FUNCTION_BLOCK FB_PROCESS_MAIN IMPLEMENTS I_PROCESS_MAIN
VAR //General
	{attribute 'instance-path'} 
  {attribute 'noinit'} 
	strInstancePath:									                      STRING;
	bInit: 												                          BOOL:=TRUE;
	strFullObjectPath: 								                      STRING;
	stEvent:											                          ST_EVENT;
	bAck:												                            BOOL;
	bNext:                                                  BOOL;
  bStop:                                                  BOOL;
END_VAR
VAR   // From FB_init	
	itfLogEvents: 										                      I_HANDLE_EVENTS;
  itfOpMode:											                        I_OP_MODE;  
  itfTimerNest1:                                          I_CLOCK; 
  itfTimerNest2:                                          I_CLOCK; 
  itfTimerNest3:                                          I_CLOCK; 
  itfTimerNest4:                                          I_CLOCK;
  itfNest1:                                               I_PROCESS_NEST1;
  itfNest2:                                               I_PROCESS_NEST2_4;
  itfNest3:                                               I_PROCESS_NEST2_4;
  itfNest4:                                               I_PROCESS_NEST2_4;
  itfLowPressurePump:                                     I_PUMP_WITH_BYPASS;
  itfOilCooler:                                           I_PUMP;
  itfBypassPump:                                          I_PUMP;
  itfLevelSwitch_AggregateTank1_Out1:                     I_BINARY_SWITCH;
  itfLevelSwitch_AggregateTank1_Out2:                     I_BINARY_SWITCH;
  itfTemperatureSwitch_AggregateTank1_Out1:               I_BINARY_SWITCH;
  itfTemperatureSwitch_AggregateTank1_Out2:               I_BINARY_SWITCH;
  itfLevelSwitch_AggregateTank2_Out1:                     I_BINARY_SWITCH;
  itfLevelSwitch_AggregateTank2_Out2:                     I_BINARY_SWITCH;
  itfLevelSwitch_AggregateTank2_Out3:                     I_BINARY_SWITCH;
  itfSwitch_AggregateFilter_Dirty:                        I_BINARY_SWITCH;  
END_VAR                                      				
VAR	// Step chain control                				
  eSeq, eLastSeq, eNextSeq:					                      E_SEQ_PROCESS; 
                  				
  //eActiveSeqState, eLastActiveSeqState:                 E_SEQ_GENERAL;
	(*
  iInternalSeqStateCase, iLastInternalSeqStateCase:       INT:=0;       
	tonDelay, tonTimeOut, tonStepTime:						          TON;
	tDelay:													                        TIME := T#100MS;
	tTimeOut:												                        TIME := T#100MS;
	tTimeOutExt:											                      TIME := T#100MS;
	bDelayActive, bTimeOutActiveQuit, bTimeOutActiveNoQuit:	BOOL;//Timer Option
	bActiveStep, bDebugAcitve, bDebugNext:					        BOOL;//Debug Option
	i:														                          INT;
 	iError:													                        INT; //ERROR-CODE                    	                   		
	listLastSteps:											                    ARRAY[0..49] OF ST_LAST_STEPS;	
	strExtraInfo:											                      STRING; 
	eStep_Type:												                      E_STEP_STATE_TYPE; 
	bDebugModeActive:										                    BOOL;   
	bWaitForBreakpoint:										                  BOOL;
	bBreakpointActive:										                  BOOL;
	bDebugResume:											                      BOOL;   
	listBreakpoint:											                    ARRAY[0..10] OF  INT;    
  *)
  i:														                            INT;
  stSeqCtrlGeneral:											                    ST_SEQ_CTRL_GEN;  
  strSeq:                                                   STRING;   	
  uiRequestId:                                              UINT;
END_VAR                                             		
VAR                                                 		
	bMethodeFromExtStarted:									                BOOL;
	bMethodeFromExtActive:									                BOOL;
	bMethodeFromExtDone:									                  BOOL;
	strTemp:												                        STRING;
END_VAR   
VAR
  udiCurrentCyclesNest1:                                  UDINT := 0;
  udiCurrentCyclesNest2:                                  UDINT := 0;
  udiCurrentCyclesNest3:                                  UDINT := 0;
  udiCurrentCyclesNest4:                                  UDINT := 0;
  udiCyclesPerLoop:                                       UDINT := 0;
  udiLoops:                                               UDINT := 0;
  uiCurrentLoop:                                          UINT := 1;
  udiResidualVal:                                         UDINT := 0;
  uiVentCount:                                            UINT;
  iOpStep:                                                INT := 0;
  bRunning:                                               BOOL;
END_VAR 
VAR // Input variables
  stERParams:                                             ST_RECIPE_ENDURANCE_RUN;
  stBPDParams:                                            ST_RECIPE_BREAK_PRESSURE;
  stLT1Params:                                            ST_RECIPE_LEAK_TEST1;
  stLT2Params:                                            ST_RECIPE_LEAK_TEST2;
END_VAR                   	
VAR_TEMP                    	
	iTemp:											                            INT;
END_VAR

// Set FBs and Interfaces ready after switch internal step
IF stSeqCtrlGeneral.iInternalSeqStateCase <> stSeqCtrlGeneral.iLastInternalSeqStateCase AND NOT stSeqCtrlGeneral.bExitSetReadyState THEN
  IF TRUE
  AND itfNest1.M_SetReady()
  AND itfNest2.M_SetReady()
  AND itfNest3.M_SetReady()
  AND itfNest4.M_SetReady()
  AND itfLowPressurePump.M_SetReady()
  AND itfOilCooler.M_SetReady()
  AND itfBypassPump.M_SetReady()
  THEN
    stSeqCtrlGeneral.bExitSetReadyState := TRUE;
  ELSE
    RETURN;
  END_IF
END_IF

stSeqCtrlGeneral.strObject:=F_CreateObjectName(strInstancePath);

// First method call
_m_SequenceManager();
//_m_SaveLastStep();

strSeq := TO_STRING(eSeq);

CASE eSeq OF 
  E_SEQ_VALVE.BASE:;
  
	E_SEQ_PROCESS.INIT: _m_Seq_INIT();
		IF TRUE
		AND (stSeqCtrlGeneral.eActiveSeqState = E_SEQ_GENERAL.DONE) 
		THEN
      eSeq := eNextSeq := E_SEQ_PROCESS.BASE;
		END_IF
		
	E_SEQ_PROCESS.SETUP:;
  
	// Process
	E_SEQ_PROCESS.ENDURANCE_RUN: _m_Seq_ENDURANCE_RUN();
    IF TRUE
		AND (stSeqCtrlGeneral.eActiveSeqState = E_SEQ_GENERAL.DONE) 
		THEN
      eSeq := eNextSeq := E_SEQ_PROCESS.BASE;
		END_IF
 
  E_SEQ_PROCESS.BREAK_PRESSURE_DET: _m_Seq_BREAK_PRESSURE_DET();
    IF TRUE
		AND (stSeqCtrlGeneral.eActiveSeqState = E_SEQ_GENERAL.DONE) 
		THEN
      eSeq := eNextSeq := E_SEQ_PROCESS.BASE;
		END_IF
    
  E_SEQ_PROCESS.LEAK_TEST_1: _m_Seq_LEAK_TEST_1();
    IF TRUE
		AND (stSeqCtrlGeneral.eActiveSeqState = E_SEQ_GENERAL.DONE) 
		THEN
      eSeq := eNextSeq := E_SEQ_PROCESS.BASE;
		END_IF
    
  E_SEQ_PROCESS.LEAK_TEST_2: _m_Seq_LEAK_TEST_2();
    IF TRUE
		AND (stSeqCtrlGeneral.eActiveSeqState = E_SEQ_GENERAL.DONE) 
		THEN
      eSeq := eNextSeq := E_SEQ_PROCESS.BASE;
		END_IF
       
  E_SEQ_PROCESS.STOP: _m_Seq_STOP();
    IF TRUE
		AND (stSeqCtrlGeneral.eActiveSeqState = E_SEQ_GENERAL.DONE) 
		THEN
      eSeq := eNextSeq := E_SEQ_PROCESS.BASE;
		END_IF
    
  E_SEQ_PROCESS.STOP_ENGINE: _m_Seq_STOP_ENGINE();
    IF TRUE
		AND (stSeqCtrlGeneral.eActiveSeqState = E_SEQ_GENERAL.DONE) 
		THEN
      eSeq := eNextSeq := E_SEQ_PROCESS.BASE;
		END_IF
    
  E_SEQ_PROCESS.ESTOP: _m_Seq_ESTOP();
    IF TRUE
		AND (stSeqCtrlGeneral.eActiveSeqState = E_SEQ_GENERAL.DONE) 
		THEN
      eSeq := eNextSeq := E_SEQ_PROCESS.BASE;
		END_IF
  
  // End
	E_SEQ_PROCESS.END:;
	E_SEQ_PROCESS.ERROR_SEQ:;	
END_CASE

strTemp:=TO_STRING(eSeq);

METHOD PRIVATE _m_DebugManager
VAR_INPUT
	iStepID: int;
END_VAR
IF TRUE
AND THIS^.stSeqCtrlGeneral.bDebugModeActive 
AND NOT THIS^.stSeqCtrlGeneral.bActiveStep
THEN


THIS^.stSeqCtrlGeneral.bBreakpointActive:=FALSE;

FOR i:=0 TO 10 DO
	
	IF TRUE
	AND iStepID=THIS^.stSeqCtrlGeneral.listBreakpoint[i] 
	AND iStepID<>0
	THEN
		EXIT;
	END_IF
END_FOR
IF (i<=10) THEN
	THIS^.stSeqCtrlGeneral.bBreakpointActive:=TRUE;
END_IF

END_IF
END_METHOD

METHOD _m_Delay : BOOL
VAR_INPUT
	DelayTime:	TIME;
END_VAR
THIS^.stSeqCtrlGeneral.bDelayActive:=TRUE;
THIS^.stSeqCtrlGeneral.tDelay:=DelayTime;
_m_Delay:=FALSE;
IF THIS^.stSeqCtrlGeneral.tonDelay.Q THEN
	_m_Delay:=TRUE;
END_IF
END_METHOD

METHOD PRIVATE _m_GeneralStepSetting : BOOL
VAR_INPUT
	StepType:			    	E_STEP_STATE_TYPE;
	InfoTextID:					STRING(20);
	EnableDebug:	   			BOOL;	
	
END_VAR
IF THIS^.stSeqCtrlGeneral.bActiveStep THEN
	THIS^.stSeqCtrlGeneral.eStep_Type:=StepType;
	THIS^.stSeqCtrlGeneral.strExtraInfo:= GenLib.F_RET_TXTLIST_ENTRY(strPortNr:='851',strID:='',strTxtLstName:=InfoTextID);
END_IF
END_METHOD

METHOD PRIVATE _m_SaveLastStep : BOOL
VAR_INPUT
END_VAR
VAR
	i: dint;
END_VAR
IF NOT THIS^.stSeqCtrlGeneral.bActiveStep THEN
	
	FOR i:=49 TO 1 BY -1 DO
			stSeqCtrlGeneral.listLastSteps[i].strStepName:=stSeqCtrlGeneral.listLastSteps[i-1].strStepName;
			stSeqCtrlGeneral.listLastSteps[i].tStepTime:=stSeqCtrlGeneral.listLastSteps[i-1].tStepTime;
			stSeqCtrlGeneral.listLastSteps[i].tDelayTime:=stSeqCtrlGeneral.listLastSteps[i-1].tDelayTime;
	END_FOR
	stSeqCtrlGeneral.listLastSteps[0].strStepName:=TO_STRING(THIS^.eSeq);
	stSeqCtrlGeneral.listLastSteps[1].tStepTime:=THIS^.stSeqCtrlGeneral.tonStepTime.ET;
	stSeqCtrlGeneral.listLastSteps[1].tStepTime:=THIS^.stSeqCtrlGeneral.tonDelay.ET;
ELSE
	stSeqCtrlGeneral.listLastSteps[0].tStepTime:=THIS^.stSeqCtrlGeneral.tonStepTime.ET;
	stSeqCtrlGeneral.listLastSteps[0].tDelayTime:=THIS^.stSeqCtrlGeneral.tonDelay.ET;	
END_IF
END_METHOD

METHOD PRIVATE _m_Seq_BREAK_PRESSURE_DET : E_SEQ_PROCESS
VAR_INPUT
END_VAR
VAR
	ActiveSeq: STRING;
END_VAR
VAR
	
END_VAR
//THIS^._m_GeneralStepSetting(StepType:=E_STEP_STATE_TYPE.INIT,
ActiveSeq := TO_STRING(THIS^.eSeq);

CASE THIS^.stSeqCtrlGeneral.eActiveSeqState OF
E_SEQ_GENERAL.READY:;

	
E_SEQ_GENERAL.EXECUTE:;
	IF TRUE
	THEN
		THIS^.stSeqCtrlGeneral.eActiveSeqState := E_SEQ_GENERAL.RESET;
	END_IF
E_SEQ_GENERAL.RESET:;
	stSeqCtrlGeneral.iInternalSeqStateCase := 0;
	IF TRUE
	THEN
		THIS^.stSeqCtrlGeneral.eActiveSeqState := E_SEQ_GENERAL.BUSY;
	END_IF
  
E_SEQ_GENERAL.BUSY:;
	CASE THIS^.stSeqCtrlGeneral.iInternalSeqStateCase OF
    0:  // check validity
      IF TRUE
      AND THIS^.stBPDParams.rMinSpeedInMmPerS > 0.1
      AND THIS^.stBPDParams.rEndPosTol > 0
      AND THIS^.stBPDParams.rIncreaseInterval > 0.1
      AND THIS^.stBPDParams.rIncreaseInterval < 10
      AND THIS^.stBPDParams.rNokLimit > 1
			THEN 
				THIS^.stSeqCtrlGeneral.iInternalSeqStateCase := 5; 
      ELSE
        THIS^.stSeqCtrlGeneral.eActiveSeqState := E_SEQ_GENERAL.ERROR; // Error step
			END_IF
      
    5:  // Start timer
      IF THIS^.itfNest1.P_EnableState THEN
        THIS^.itfTimerNest1.M_StartTimer();
			END_IF
      THIS^.stSeqCtrlGeneral.iInternalSeqStateCase := 10;

    10:  // Nest 1 vent cylinder
      IF TRUE
      AND THIS^.itfLowPressurePump.M_Bypass(bEnable:= TRUE)
			AND THIS^.itfNest1.M_VentCylinder(uiVentCount:= THIS^.stBPDParams.uiVentCycles)
			THEN 
				THIS^.stSeqCtrlGeneral.iInternalSeqStateCase := 20; 
			END_IF
      
    20:  // Low pressure pump off
      IF TRUE  
      AND THIS^.itfLowPressurePump.M_Off()
			THEN 
				THIS^.stSeqCtrlGeneral.iInternalSeqStateCase := 30; 
			END_IF
      
    30:  // Nest 1 determinate stroke length
      IF TRUE 
			AND THIS^.itfNest1.M_MeasureStrokeLength()
			THEN 
				THIS^.stSeqCtrlGeneral.iInternalSeqStateCase := 40; 
			END_IF
      
    40:  // Nest 1 endurance run
      IF TRUE 
			AND THIS^.itfNest1.M_BreakPressureDet(stBreakPressureParams:= THIS^.stBPDParams)
			THEN 
				THIS^.stSeqCtrlGeneral.iInternalSeqStateCase := 1000; // Exit step
			END_IF
      
    1000: // Exit step
      IF TRUE 
      AND THIS^.itfTimerNest1.M_StopTimer()
			THEN 
				THIS^.stSeqCtrlGeneral.iInternalSeqStateCase := 9999; 
			END_IF
      
	ELSE
		THIS^.stSeqCtrlGeneral.eActiveSeqState := E_SEQ_GENERAL.DONE;  
	END_CASE
	THIS^.stSeqCtrlGeneral.strExtraInfo := CONCAT('Internal state: ', TO_STRING(THIS^.stSeqCtrlGeneral.iInternalSeqStateCase));
E_SEQ_GENERAL.DONE:;
E_SEQ_GENERAL.ERROR:;
E_SEQ_GENERAL.TIME_OUT:; 

IF TRUE
AND THIS^.stSeqCtrlGeneral.bTimeOutActiveQuit 
THEN
  THIS^.stSeqCtrlGeneral.strExtraInfo := 'Bitte quittieren und erneut testen';
  IF TRUE
  //AND itfOpMode.P_QUIT
  THEN
    THIS^.stSeqCtrlGeneral.eActiveSeqState := E_SEQ_GENERAL.EXECUTE;
	END_IF
  
END_IF

ELSE
  THIS^.stSeqCtrlGeneral.eActiveSeqState := E_SEQ_GENERAL.ERROR;
END_CASE
END_METHOD

METHOD PRIVATE _m_Seq_ENDURANCE_RUN : E_SEQ_PROCESS
VAR_INPUT
END_VAR
VAR
	ActiveSeq:                      STRING;
END_VAR
//THIS^._m_GeneralStepSetting(StepType:=E_STEP_STATE_TYPE.INIT,
ActiveSeq := TO_STRING(THIS^.eSeq);

CASE THIS^.stSeqCtrlGeneral.eActiveSeqState OF
E_SEQ_GENERAL.READY:;

	
E_SEQ_GENERAL.EXECUTE:;
	IF TRUE
	THEN
		THIS^.stSeqCtrlGeneral.eActiveSeqState := E_SEQ_GENERAL.RESET;
	END_IF
E_SEQ_GENERAL.RESET:;
	stSeqCtrlGeneral.iInternalSeqStateCase := 0;
	IF TRUE
	THEN
    THIS^.udiCyclesPerLoop := THIS^.stERParams.udiCycles;
    THIS^.udiLoops := 1;
    THIS^.uiCurrentLoop := 1;
    THIS^.udiResidualVal := 0;
		THIS^.stSeqCtrlGeneral.eActiveSeqState := E_SEQ_GENERAL.BUSY;
	END_IF
  
E_SEQ_GENERAL.BUSY:;
	CASE THIS^.stSeqCtrlGeneral.iInternalSeqStateCase OF
    0:  // check validity
      IF TRUE
      AND THIS^.stERParams.rSpeedA > 1
      AND THIS^.stERParams.rSpeedB > 1
      AND THIS^.stERParams.rTurningPointHP > 0
      AND THIS^.stERParams.rTurningPointWP > 0
      AND THIS^.stERParams.rWorkForceA > 0.1
      AND THIS^.stERParams.rWorkForceB > 0.1
      AND THIS^.stERParams.udiCycles > 1
			THEN 
				THIS^.stSeqCtrlGeneral.iInternalSeqStateCase := 5; 
      ELSE
        THIS^.stSeqCtrlGeneral.eActiveSeqState := E_SEQ_GENERAL.ERROR; // Error step
			END_IF
      
    5:  // Start timer
      IF THIS^.itfNest1.P_EnableState THEN
        THIS^.itfTimerNest1.M_StartTimer();
			END_IF
      IF THIS^.itfNest2.P_EnableState THEN
        THIS^.itfTimerNest2.M_StartTimer();
			END_IF
      IF THIS^.itfNest3.P_EnableState THEN
        THIS^.itfTimerNest3.M_StartTimer();
			END_IF
      IF THIS^.itfNest4.P_EnableState THEN
        THIS^.itfTimerNest4.M_StartTimer();
			END_IF
      THIS^.stSeqCtrlGeneral.iInternalSeqStateCase := 10;

    10:  // Nest 1-4 vent cylinder
      IF TRUE
      AND THIS^.itfLowPressurePump.M_Bypass(bEnable:= TRUE)
			AND THIS^.itfNest1.M_VentCylinder(uiVentCount:= THIS^.stERParams.uiVentCycles)
      AND THIS^.itfNest2.M_VentCylinder(uiVentCount:= THIS^.stERParams.uiVentCycles)
      AND THIS^.itfNest3.M_VentCylinder(uiVentCount:= THIS^.stERParams.uiVentCycles)
      AND THIS^.itfNest4.M_VentCylinder(uiVentCount:= THIS^.stERParams.uiVentCycles)
			THEN 
				THIS^.stSeqCtrlGeneral.iInternalSeqStateCase := 20; 
			END_IF
      
    20:  // Nest 1-4 determinate stroke length
      IF TRUE  
      AND THIS^.itfLowPressurePump.M_On()
			AND THIS^.itfNest1.M_MeasureStrokeLength()
      AND THIS^.itfNest2.M_MeasureStrokeLength()
      AND THIS^.itfNest3.M_MeasureStrokeLength()
      AND THIS^.itfNest4.M_MeasureStrokeLength()
			THEN 
				THIS^.stSeqCtrlGeneral.iInternalSeqStateCase := 30; 
			END_IF
      
    30:  // Nest 1 determinate max speed (VMAX)
      IF TRUE  
			AND THIS^.itfNest1.M_MaxSpeedRecord(stEnduranceRunParams:= THIS^.stERParams)
			THEN 
        IF TRUE
        AND (THIS^.stERParams.rSpeedA > THIS^.itfNest1.P_MaxSpeedInMmPerSWP * THIS^.itfNest1.P_SpeedEfficiencyFactor
        OR THIS^.stERParams.rSpeedB > THIS^.itfNest1.P_MaxSpeedInMmPerSHP * THIS^.itfNest1.P_SpeedEfficiencyFactor) 
        THEN
          THIS^.itfNest2.M_SetEnableState(bEnable:= FALSE);
          THIS^.itfNest3.M_SetEnableState(bEnable:= FALSE);
          THIS^.itfNest4.M_SetEnableState(bEnable:= FALSE);
          THIS^.itfTimerNest2.M_StopTimer();
          THIS^.itfTimerNest3.M_StopTimer();
          THIS^.itfTimerNest4.M_StopTimer();
				END_IF
				THIS^.stSeqCtrlGeneral.iInternalSeqStateCase := 40; 
			END_IF
      
    40:  // Calc loops and cycles
      IF TRUE
      AND THIS^.stERParams.bEnableLeakTest1
      THEN
        THIS^.udiCyclesPerLoop := THIS^.stERParams.udiLT1_Interval;
        THIS^.udiLoops := THIS^.stERParams.udiCycles / THIS^.stERParams.udiLT1_Interval - 1;
        THIS^.udiResidualVal := THIS^.stERParams.udiCycles - THIS^.udiLoops * THIS^.udiCyclesPerLoop;
			END_IF
      THIS^.stSeqCtrlGeneral.iInternalSeqStateCase := 50; 
      
    50:  // Nest 1 endurance run
      IF TRUE 
      AND THIS^.itfLowPressurePump.M_Bypass(bEnable:= FALSE)
			AND THIS^.itfNest1.M_EnduranceRun(udiCycles:= THIS^.udiCyclesPerLoop, stEnduranceRunParams:= THIS^.stERParams)
      AND THIS^.itfNest2.M_EnduranceRun(udiCycles:= THIS^.udiCyclesPerLoop, stEnduranceRunParams:= THIS^.stERParams)
      AND THIS^.itfNest3.M_EnduranceRun(udiCycles:= THIS^.udiCyclesPerLoop, stEnduranceRunParams:= THIS^.stERParams)
      AND THIS^.itfNest4.M_EnduranceRun(udiCycles:= THIS^.udiCyclesPerLoop, stEnduranceRunParams:= THIS^.stERParams)
			THEN 
        THIS^.uiCurrentLoop := THIS^.uiCurrentLoop + 1;
				THIS^.stSeqCtrlGeneral.iInternalSeqStateCase := 60; 
			END_IF
      THIS^.udiCurrentCyclesNest1 := THIS^.udiCyclesPerLoop * (THIS^.uiCurrentLoop - 1) + THIS^.itfNest1.P_CurrentCycle;
      THIS^.udiCurrentCyclesNest2 := THIS^.udiCyclesPerLoop * (THIS^.uiCurrentLoop - 1) + THIS^.itfNest2.P_CurrentCycle;
      THIS^.udiCurrentCyclesNest3 := THIS^.udiCyclesPerLoop * (THIS^.uiCurrentLoop - 1) + THIS^.itfNest3.P_CurrentCycle;
      THIS^.udiCurrentCyclesNest4 := THIS^.udiCyclesPerLoop * (THIS^.uiCurrentLoop - 1) + THIS^.itfNest4.P_CurrentCycle;
      
    60:  // Choice step
      IF TRUE
      AND THIS^.stERParams.bEnableLeakTest1
      THEN
        THIS^.stSeqCtrlGeneral.iInternalSeqStateCase := 70; 
      ELSE
        THIS^.stSeqCtrlGeneral.iInternalSeqStateCase := 1000; // Exit seq
			END_IF
      
    70:  // Leak test 1
      IF TRUE
      AND THIS^.itfNest1.M_LeakTest1(stLeakTest1Params:= THIS^.stERParams.stLT1_Params)
      AND THIS^.itfNest2.M_LeakTest1(stLeakTest1Params:= THIS^.stERParams.stLT1_Params)
      AND THIS^.itfNest3.M_LeakTest1(stLeakTest1Params:= THIS^.stERParams.stLT1_Params)
      AND THIS^.itfNest4.M_LeakTest1(stLeakTest1Params:= THIS^.stERParams.stLT1_Params)
      THEN
        THIS^.stSeqCtrlGeneral.iInternalSeqStateCase := 80;
      END_IF
      
    80:  // Choice step
      IF TRUE
      AND THIS^.uiCurrentLoop <= THIS^.udiLoops
      THEN
        THIS^.stSeqCtrlGeneral.iInternalSeqStateCase := 50; // Jump backward
      ELSE
        THIS^.stSeqCtrlGeneral.iInternalSeqStateCase := 90;
      END_IF
      
    90:  // Last endurance run loop
      IF TRUE 
      AND THIS^.itfLowPressurePump.M_Bypass(bEnable:= FALSE)
			AND THIS^.itfNest1.M_EnduranceRun(udiCycles:= THIS^.udiCyclesPerLoop + THIS^.udiResidualVal, stEnduranceRunParams:= THIS^.stERParams)
      AND THIS^.itfNest2.M_EnduranceRun(udiCycles:= THIS^.udiCyclesPerLoop + THIS^.udiResidualVal, stEnduranceRunParams:= THIS^.stERParams)
      AND THIS^.itfNest3.M_EnduranceRun(udiCycles:= THIS^.udiCyclesPerLoop + THIS^.udiResidualVal, stEnduranceRunParams:= THIS^.stERParams)
      AND THIS^.itfNest4.M_EnduranceRun(udiCycles:= THIS^.udiCyclesPerLoop + THIS^.udiResidualVal, stEnduranceRunParams:= THIS^.stERParams)
			THEN 
				THIS^.stSeqCtrlGeneral.iInternalSeqStateCase := 1000; 
			END_IF
      
    1000:  // Enable low pressure circuit bypass
      IF TRUE 
      AND THIS^.itfLowPressurePump.M_Bypass(bEnable:= TRUE)
			THEN 
				THIS^.stSeqCtrlGeneral.iInternalSeqStateCase := 1010; 
			END_IF
      
    1010: // Exit seq
      IF TRUE 
      AND THIS^.itfTimerNest1.M_StopTimer()
      AND THIS^.itfTimerNest2.M_StopTimer()
      AND THIS^.itfTimerNest3.M_StopTimer()
      AND THIS^.itfTimerNest4.M_StopTimer()
			THEN 
				THIS^.stSeqCtrlGeneral.iInternalSeqStateCase := 9999; 
			END_IF
      
	ELSE
		THIS^.stSeqCtrlGeneral.eActiveSeqState := E_SEQ_GENERAL.DONE;  
	END_CASE
	THIS^.stSeqCtrlGeneral.strExtraInfo := CONCAT('Internal state: ', TO_STRING(THIS^.stSeqCtrlGeneral.iInternalSeqStateCase));
E_SEQ_GENERAL.DONE:;
E_SEQ_GENERAL.ERROR:;
E_SEQ_GENERAL.TIME_OUT:; 

IF TRUE
AND THIS^.stSeqCtrlGeneral.bTimeOutActiveQuit 
THEN
  THIS^.stSeqCtrlGeneral.strExtraInfo := 'Bitte quittieren und erneut testen';
  IF TRUE
  //AND itfOpMode.P_QUIT
  THEN
    THIS^.stSeqCtrlGeneral.eActiveSeqState := E_SEQ_GENERAL.EXECUTE;
	END_IF
  
END_IF

ELSE
  THIS^.stSeqCtrlGeneral.eActiveSeqState := E_SEQ_GENERAL.ERROR;
END_CASE
END_METHOD

METHOD PRIVATE _m_Seq_ESTOP : E_SEQ_PROCESS
VAR_INPUT
END_VAR
VAR
	ActiveSeq: STRING;
END_VAR
VAR
	
END_VAR
//THIS^._m_GeneralStepSetting(StepType:=E_STEP_STATE_TYPE.INIT,
ActiveSeq := TO_STRING(THIS^.eSeq);

CASE THIS^.stSeqCtrlGeneral.eActiveSeqState OF
E_SEQ_GENERAL.READY:;

	
E_SEQ_GENERAL.EXECUTE:;
	IF TRUE
	THEN
		THIS^.stSeqCtrlGeneral.eActiveSeqState := E_SEQ_GENERAL.RESET;
	END_IF
E_SEQ_GENERAL.RESET:;
	stSeqCtrlGeneral.iInternalSeqStateCase := 0;
	IF TRUE
	THEN
		THIS^.stSeqCtrlGeneral.eActiveSeqState := E_SEQ_GENERAL.BUSY;
	END_IF
  
E_SEQ_GENERAL.BUSY:;
	CASE THIS^.stSeqCtrlGeneral.iInternalSeqStateCase OF
    0:  // Nest 1 stop and enable low pressure pump bypass
      IF TRUE 
			AND THIS^.itfNest1.M_Stop()
      AND THIS^.itfLowPressurePump.M_Bypass(bEnable:= TRUE)
			THEN 
				THIS^.stSeqCtrlGeneral.iInternalSeqStateCase := 10; 
			END_IF
      
    10:  // Nest 2-4 stop
      IF TRUE 
			AND THIS^.itfNest2.M_Stop()
			AND THIS^.itfNest3.M_Stop()
			AND THIS^.itfNest4.M_Stop()
			THEN 
				THIS^.stSeqCtrlGeneral.iInternalSeqStateCase := 20; 
			END_IF
      
    20:  // Nest 1 stop engine
      IF TRUE 
			AND THIS^.itfNest1.M_StopEngine()
			THEN 
				THIS^.stSeqCtrlGeneral.iInternalSeqStateCase := 30; 
			END_IF
      
    30:  // Nest 2-4 stop engine
      IF TRUE 
			AND THIS^.itfNest2.M_StopEngine()
			AND THIS^.itfNest3.M_StopEngine()
			AND THIS^.itfNest4.M_StopEngine()
			THEN 
				THIS^.stSeqCtrlGeneral.iInternalSeqStateCase := 1000; 
			END_IF
      
    1000: // Exit step
      IF TRUE
      AND THIS^.itfTimerNest1.M_StopTimer()
      AND THIS^.itfTimerNest2.M_StopTimer()
      AND THIS^.itfTimerNest3.M_StopTimer()
      AND THIS^.itfTimerNest4.M_StopTimer()
			THEN 
				THIS^.stSeqCtrlGeneral.iInternalSeqStateCase := 9999; 
			END_IF
      
	ELSE
		THIS^.stSeqCtrlGeneral.eActiveSeqState := E_SEQ_GENERAL.DONE;  
	END_CASE
	THIS^.stSeqCtrlGeneral.strExtraInfo := CONCAT('Internal state: ', TO_STRING(THIS^.stSeqCtrlGeneral.iInternalSeqStateCase));
E_SEQ_GENERAL.DONE:;
E_SEQ_GENERAL.ERROR:;
E_SEQ_GENERAL.TIME_OUT:; 

IF TRUE
AND THIS^.stSeqCtrlGeneral.bTimeOutActiveQuit 
THEN
  THIS^.stSeqCtrlGeneral.strExtraInfo := 'Bitte quittieren und erneut testen';
  IF TRUE
  //AND itfOpMode.P_QUIT
  THEN
    THIS^.stSeqCtrlGeneral.eActiveSeqState := E_SEQ_GENERAL.EXECUTE;
	END_IF
  
END_IF

ELSE
  THIS^.stSeqCtrlGeneral.eActiveSeqState := E_SEQ_GENERAL.ERROR;
END_CASE
END_METHOD

METHOD PRIVATE _m_Seq_INIT : E_SEQ_PROCESS
VAR_INPUT
END_VAR
VAR
	ActiveSeq: STRING;
END_VAR
VAR
	
END_VAR
//THIS^._m_GeneralStepSetting(StepType:=E_STEP_STATE_TYPE.INIT,
ActiveSeq := TO_STRING(THIS^.eSeq);

CASE THIS^.stSeqCtrlGeneral.eActiveSeqState OF
E_SEQ_GENERAL.READY:;

	
E_SEQ_GENERAL.EXECUTE:;
	IF TRUE
	THEN
		THIS^.stSeqCtrlGeneral.eActiveSeqState := E_SEQ_GENERAL.RESET;
	END_IF
E_SEQ_GENERAL.RESET:;
	stSeqCtrlGeneral.iInternalSeqStateCase := 0;
	IF TRUE
	THEN
		THIS^.stSeqCtrlGeneral.eActiveSeqState := E_SEQ_GENERAL.BUSY;
	END_IF
  
E_SEQ_GENERAL.BUSY:;
	CASE THIS^.stSeqCtrlGeneral.iInternalSeqStateCase OF
    0:  // Nest 1 reset
      IF TRUE 
      AND THIS^.itfTimerNest1.M_StartTimer()
			AND THIS^.itfNest1.M_Reset()
			THEN 
				THIS^.stSeqCtrlGeneral.iInternalSeqStateCase := 10; 
			END_IF
      
    10: // Nest 2 reset
      IF TRUE 
      AND THIS^.itfTimerNest2.M_StartTimer()
			AND THIS^.itfNest2.M_Reset()
			THEN 
				THIS^.stSeqCtrlGeneral.iInternalSeqStateCase := 20; 
			END_IF
      
    20: // Nest 3 reset
      IF TRUE 
      AND THIS^.itfTimerNest3.M_StartTimer()
			AND THIS^.itfNest3.M_Reset()
			THEN 
				THIS^.stSeqCtrlGeneral.iInternalSeqStateCase := 30; 
			END_IF
      
    30: // Nest 4 reset
      IF TRUE 
      AND THIS^.itfTimerNest4.M_StartTimer()
			AND THIS^.itfNest4.M_Reset()
			THEN 
				THIS^.stSeqCtrlGeneral.iInternalSeqStateCase := 40; 
			END_IF
      
    40: // Low pressure pump reset
      IF TRUE 
			AND THIS^.itfLowPressurePump.M_Off()
			THEN 
				THIS^.stSeqCtrlGeneral.iInternalSeqStateCase := 50; 
			END_IF
      
    50: // Low pressure pump reset
      IF TRUE 
			AND THIS^.itfLowPressurePump.M_Bypass(bEnable:= TRUE)
			THEN 
				THIS^.stSeqCtrlGeneral.iInternalSeqStateCase := 60; 
			END_IF
      
    60: // Low pressure pump reset
      IF TRUE 
			AND THIS^.itfLowPressurePump.M_On()
			THEN 
				THIS^.stSeqCtrlGeneral.iInternalSeqStateCase := 1000; 
			END_IF
      
    1000: // Exit step
      IF TRUE
      AND THIS^.itfTimerNest1.M_StopTimer()
      AND THIS^.itfTimerNest2.M_StopTimer()
      AND THIS^.itfTimerNest3.M_StopTimer()
      AND THIS^.itfTimerNest4.M_StopTimer()
			THEN 
				THIS^.stSeqCtrlGeneral.iInternalSeqStateCase := 9999; 
			END_IF
      
	ELSE
		THIS^.stSeqCtrlGeneral.eActiveSeqState := E_SEQ_GENERAL.DONE;  
	END_CASE
	THIS^.stSeqCtrlGeneral.strExtraInfo := CONCAT('Internal state: ', TO_STRING(THIS^.stSeqCtrlGeneral.iInternalSeqStateCase));
E_SEQ_GENERAL.DONE:;
E_SEQ_GENERAL.ERROR:;
E_SEQ_GENERAL.TIME_OUT:; 

IF TRUE
AND THIS^.stSeqCtrlGeneral.bTimeOutActiveQuit 
THEN
  THIS^.stSeqCtrlGeneral.strExtraInfo := 'Bitte quittieren und erneut testen';
  IF TRUE
  //AND itfOpMode.P_QUIT
  THEN
    THIS^.stSeqCtrlGeneral.eActiveSeqState := E_SEQ_GENERAL.EXECUTE;
	END_IF
  
END_IF

ELSE
  THIS^.stSeqCtrlGeneral.eActiveSeqState := E_SEQ_GENERAL.ERROR;
END_CASE
END_METHOD

METHOD PRIVATE _m_Seq_LEAK_TEST_1 : E_SEQ_PROCESS
VAR_INPUT
END_VAR
VAR
	ActiveSeq: STRING;
END_VAR
VAR
	
END_VAR
//THIS^._m_GeneralStepSetting(StepType:=E_STEP_STATE_TYPE.INIT,
ActiveSeq := TO_STRING(THIS^.eSeq);

CASE THIS^.stSeqCtrlGeneral.eActiveSeqState OF
E_SEQ_GENERAL.READY:;

	
E_SEQ_GENERAL.EXECUTE:;
	IF TRUE
	THEN
		THIS^.stSeqCtrlGeneral.eActiveSeqState := E_SEQ_GENERAL.RESET;
	END_IF
E_SEQ_GENERAL.RESET:;
	stSeqCtrlGeneral.iInternalSeqStateCase := 0;
	IF TRUE
	THEN
		THIS^.stSeqCtrlGeneral.eActiveSeqState := E_SEQ_GENERAL.BUSY;
	END_IF
  
E_SEQ_GENERAL.BUSY:;
	CASE THIS^.stSeqCtrlGeneral.iInternalSeqStateCase OF
    0:  // check validity
      IF TRUE
      AND THIS^.stLT1Params.rDistanceBeforeEndPosHP > 0
      AND THIS^.stLT1Params.rDistanceBeforeEndPosWP > 0
      AND THIS^.stLT1Params.rLoadForceA > 0.1
      AND THIS^.stLT1Params.rLoadForceA > 0.1
      AND THIS^.stLT1Params.rNokLimit > 0.05
      AND THIS^.stLT1Params.rRestDelay > 0
      AND THIS^.stLT1Params.udiDurationPerTest > 0
			THEN 
				THIS^.stSeqCtrlGeneral.iInternalSeqStateCase := 5; 
      ELSE
        THIS^.stSeqCtrlGeneral.eActiveSeqState := E_SEQ_GENERAL.ERROR; // Error step
			END_IF
      
    5:  // Start timer
      IF THIS^.itfNest1.P_EnableState THEN
        THIS^.itfTimerNest1.M_StartTimer();
			END_IF
      IF THIS^.itfNest2.P_EnableState THEN
        THIS^.itfTimerNest2.M_StartTimer();
			END_IF
      IF THIS^.itfNest3.P_EnableState THEN
        THIS^.itfTimerNest3.M_StartTimer();
			END_IF
      IF THIS^.itfNest4.P_EnableState THEN
        THIS^.itfTimerNest4.M_StartTimer();
			END_IF
      THIS^.stSeqCtrlGeneral.iInternalSeqStateCase := 10;

    10:  // Nest 1 vent cylinder
      IF TRUE
      AND THIS^.itfLowPressurePump.M_Bypass(bEnable:= TRUE)
			AND THIS^.itfNest1.M_VentCylinder(uiVentCount:= THIS^.stLT1Params.uiVentCycles)
      AND THIS^.itfNest2.M_VentCylinder(uiVentCount:= THIS^.stLT1Params.uiVentCycles)
      AND THIS^.itfNest3.M_VentCylinder(uiVentCount:= THIS^.stLT1Params.uiVentCycles)
      AND THIS^.itfNest4.M_VentCylinder(uiVentCount:= THIS^.stLT1Params.uiVentCycles)
			THEN 
				THIS^.stSeqCtrlGeneral.iInternalSeqStateCase := 20; 
			END_IF
      
    20:  // Nest 1 determinate stroke length
      IF TRUE  
      AND THIS^.itfLowPressurePump.M_Off()
			AND THIS^.itfNest1.M_MeasureStrokeLength()
      AND THIS^.itfNest2.M_MeasureStrokeLength()
      AND THIS^.itfNest3.M_MeasureStrokeLength()
      AND THIS^.itfNest4.M_MeasureStrokeLength()
			THEN 
				THIS^.stSeqCtrlGeneral.iInternalSeqStateCase := 30; 
			END_IF
      
    30:  // Nest 1 endurance run
      IF TRUE 
			AND THIS^.itfNest1.M_LeakTest1(stLeakTest1Params:= THIS^.stLT1Params)
      AND THIS^.itfNest2.M_LeakTest1(stLeakTest1Params:= THIS^.stLT1Params)
      AND THIS^.itfNest3.M_LeakTest1(stLeakTest1Params:= THIS^.stLT1Params)
      AND THIS^.itfNest4.M_LeakTest1(stLeakTest1Params:= THIS^.stLT1Params)
			THEN 
				THIS^.stSeqCtrlGeneral.iInternalSeqStateCase := 1000; 
			END_IF
      
    1000: // Exit step
      IF TRUE
      AND THIS^.itfTimerNest1.M_StopTimer()
      AND THIS^.itfTimerNest2.M_StopTimer()
      AND THIS^.itfTimerNest3.M_StopTimer()
      AND THIS^.itfTimerNest4.M_StopTimer()
			THEN 
				THIS^.stSeqCtrlGeneral.iInternalSeqStateCase := 9999; 
			END_IF
      
	ELSE
		THIS^.stSeqCtrlGeneral.eActiveSeqState := E_SEQ_GENERAL.DONE;  
	END_CASE
	THIS^.stSeqCtrlGeneral.strExtraInfo := CONCAT('Internal state: ', TO_STRING(THIS^.stSeqCtrlGeneral.iInternalSeqStateCase));
E_SEQ_GENERAL.DONE:;
E_SEQ_GENERAL.ERROR:;
E_SEQ_GENERAL.TIME_OUT:; 

IF TRUE
AND THIS^.stSeqCtrlGeneral.bTimeOutActiveQuit 
THEN
  THIS^.stSeqCtrlGeneral.strExtraInfo := 'Bitte quittieren und erneut testen';
  IF TRUE
  //AND itfOpMode.P_QUIT
  THEN
    THIS^.stSeqCtrlGeneral.eActiveSeqState := E_SEQ_GENERAL.EXECUTE;
	END_IF
  
END_IF

ELSE
  THIS^.stSeqCtrlGeneral.eActiveSeqState := E_SEQ_GENERAL.ERROR;
END_CASE
END_METHOD

METHOD PRIVATE _m_Seq_LEAK_TEST_2 : E_SEQ_PROCESS
VAR_INPUT
END_VAR
VAR
	ActiveSeq: STRING;
END_VAR
VAR
	
END_VAR
//THIS^._m_GeneralStepSetting(StepType:=E_STEP_STATE_TYPE.INIT,
ActiveSeq := TO_STRING(THIS^.eSeq);

CASE THIS^.stSeqCtrlGeneral.eActiveSeqState OF
E_SEQ_GENERAL.READY:;

	
E_SEQ_GENERAL.EXECUTE:;
	IF TRUE
	THEN
		THIS^.stSeqCtrlGeneral.eActiveSeqState := E_SEQ_GENERAL.RESET;
	END_IF
E_SEQ_GENERAL.RESET:;
	stSeqCtrlGeneral.iInternalSeqStateCase := 0;
	IF TRUE
	THEN
		THIS^.stSeqCtrlGeneral.eActiveSeqState := E_SEQ_GENERAL.BUSY;
	END_IF
  
E_SEQ_GENERAL.BUSY:;
	CASE THIS^.stSeqCtrlGeneral.iInternalSeqStateCase OF
    0:  // check validity
      IF TRUE
      AND THIS^.stLT2Params.rLoadForceA > 0.1
      AND THIS^.stLT2Params.rLoadForceA > 0.1
      AND THIS^.stLT2Params.rNokLimit > 0.05
      AND THIS^.stLT2Params.rRestDelay > 0
      AND THIS^.stLT2Params.udiDurationPerTest > 0
			THEN 
				THIS^.stSeqCtrlGeneral.iInternalSeqStateCase := 5; 
      ELSE
        THIS^.stSeqCtrlGeneral.eActiveSeqState := E_SEQ_GENERAL.ERROR; // Error step
			END_IF
      
    5:  // Start timer
      IF THIS^.itfNest1.P_EnableState THEN
        THIS^.itfTimerNest1.M_StartTimer();
			END_IF
      THIS^.stSeqCtrlGeneral.iInternalSeqStateCase := 10;

    10:  // Nest 1 vent cylinder
      IF TRUE
      AND THIS^.itfLowPressurePump.M_Bypass(bEnable:= TRUE)
			AND THIS^.itfNest1.M_VentCylinder(uiVentCount:= THIS^.stLT2Params.uiVentCycles)
			THEN 
				THIS^.stSeqCtrlGeneral.iInternalSeqStateCase := 20; 
			END_IF
      
    20:  // Nest 1 determinate stroke length
      IF TRUE  
      AND THIS^.itfLowPressurePump.M_Off()
			AND THIS^.itfNest1.M_MeasureStrokeLength()
			THEN 
				THIS^.stSeqCtrlGeneral.iInternalSeqStateCase := 30; 
			END_IF
      
    30:  // Nest 1 endurance run
      IF TRUE 
			AND THIS^.itfNest1.M_LeakTest2(stLeakTest2Params:= THIS^.stLT2Params)
			THEN 
				THIS^.stSeqCtrlGeneral.iInternalSeqStateCase := 1000; 
			END_IF
      
    1000: // Exit step
      IF TRUE
      AND THIS^.itfTimerNest1.M_StopTimer()
			THEN 
				THIS^.stSeqCtrlGeneral.iInternalSeqStateCase := 9999; 
			END_IF
      
	ELSE
		THIS^.stSeqCtrlGeneral.eActiveSeqState := E_SEQ_GENERAL.DONE;  
	END_CASE
	THIS^.stSeqCtrlGeneral.strExtraInfo := CONCAT('Internal state: ', TO_STRING(THIS^.stSeqCtrlGeneral.iInternalSeqStateCase));
E_SEQ_GENERAL.DONE:;
E_SEQ_GENERAL.ERROR:;
E_SEQ_GENERAL.TIME_OUT:; 

IF TRUE
AND THIS^.stSeqCtrlGeneral.bTimeOutActiveQuit 
THEN
  THIS^.stSeqCtrlGeneral.strExtraInfo := 'Bitte quittieren und erneut testen';
  IF TRUE
  //AND itfOpMode.P_QUIT
  THEN
    THIS^.stSeqCtrlGeneral.eActiveSeqState := E_SEQ_GENERAL.EXECUTE;
	END_IF
  
END_IF

ELSE
  THIS^.stSeqCtrlGeneral.eActiveSeqState := E_SEQ_GENERAL.ERROR;
END_CASE
END_METHOD

METHOD PRIVATE _m_Seq_STOP : E_SEQ_PROCESS
VAR_INPUT
END_VAR
VAR
	ActiveSeq: STRING;
END_VAR
VAR
	
END_VAR
//THIS^._m_GeneralStepSetting(StepType:=E_STEP_STATE_TYPE.INIT,
ActiveSeq := TO_STRING(THIS^.eSeq);

CASE THIS^.stSeqCtrlGeneral.eActiveSeqState OF
E_SEQ_GENERAL.READY:;

	
E_SEQ_GENERAL.EXECUTE:;
	IF TRUE
	THEN
		THIS^.stSeqCtrlGeneral.eActiveSeqState := E_SEQ_GENERAL.RESET;
	END_IF
E_SEQ_GENERAL.RESET:;
	stSeqCtrlGeneral.iInternalSeqStateCase := 0;
	IF TRUE
	THEN
		THIS^.stSeqCtrlGeneral.eActiveSeqState := E_SEQ_GENERAL.BUSY;
	END_IF
  
E_SEQ_GENERAL.BUSY:;
	CASE THIS^.stSeqCtrlGeneral.iInternalSeqStateCase OF
    0:  // Nest 1 stop and low pressure pump bypass
      IF TRUE 
			AND THIS^.itfNest1.M_Stop()
      AND THIS^.itfLowPressurePump.M_Bypass(bEnable:= TRUE)
			THEN 
				THIS^.stSeqCtrlGeneral.iInternalSeqStateCase := 10; 
			END_IF
      
    10:  // Nest 2-4 stop
      IF TRUE 
			AND THIS^.itfNest2.M_Stop()
			AND THIS^.itfNest3.M_Stop()
			AND THIS^.itfNest4.M_Stop()
			THEN 
				THIS^.stSeqCtrlGeneral.iInternalSeqStateCase := 1000; 
			END_IF
      
    1000: // Exit step
      IF TRUE
      AND THIS^.itfTimerNest1.M_StopTimer()
      AND THIS^.itfTimerNest2.M_StopTimer()
      AND THIS^.itfTimerNest3.M_StopTimer()
      AND THIS^.itfTimerNest4.M_StopTimer()
			THEN 
				THIS^.stSeqCtrlGeneral.iInternalSeqStateCase := 9999; 
			END_IF
      
	ELSE
		THIS^.stSeqCtrlGeneral.eActiveSeqState := E_SEQ_GENERAL.DONE;  
	END_CASE
	THIS^.stSeqCtrlGeneral.strExtraInfo := CONCAT('Internal state: ', TO_STRING(THIS^.stSeqCtrlGeneral.iInternalSeqStateCase));
E_SEQ_GENERAL.DONE:;
E_SEQ_GENERAL.ERROR:;
E_SEQ_GENERAL.TIME_OUT:; 

IF TRUE
AND THIS^.stSeqCtrlGeneral.bTimeOutActiveQuit 
THEN
  THIS^.stSeqCtrlGeneral.strExtraInfo := 'Bitte quittieren und erneut testen';
  IF TRUE
  //AND itfOpMode.P_QUIT
  THEN
    THIS^.stSeqCtrlGeneral.eActiveSeqState := E_SEQ_GENERAL.EXECUTE;
	END_IF
  
END_IF

ELSE
  THIS^.stSeqCtrlGeneral.eActiveSeqState := E_SEQ_GENERAL.ERROR;
END_CASE
END_METHOD

METHOD PRIVATE _m_Seq_STOP_ENGINE : E_SEQ_PROCESS
VAR_INPUT
END_VAR
VAR
	ActiveSeq: STRING;
END_VAR
VAR
	
END_VAR
//THIS^._m_GeneralStepSetting(StepType:=E_STEP_STATE_TYPE.INIT,
ActiveSeq := TO_STRING(THIS^.eSeq);

CASE THIS^.stSeqCtrlGeneral.eActiveSeqState OF
E_SEQ_GENERAL.READY:;

	
E_SEQ_GENERAL.EXECUTE:;
	IF TRUE
	AND _m_Delay(T#1S)
	THEN
		THIS^.stSeqCtrlGeneral.eActiveSeqState := E_SEQ_GENERAL.RESET;
	END_IF
E_SEQ_GENERAL.RESET:;
	stSeqCtrlGeneral.iInternalSeqStateCase := 0;
  
	IF TRUE
	THEN
		THIS^.stSeqCtrlGeneral.eActiveSeqState := E_SEQ_GENERAL.BUSY;
	END_IF
E_SEQ_GENERAL.BUSY:;
	CASE THIS^.stSeqCtrlGeneral.iInternalSeqStateCase OF
		0:  // Nest 1 engine stop
      IF TRUE 
			AND THIS^.itfNest1.M_StopEngine()
			THEN 
				THIS^.stSeqCtrlGeneral.iInternalSeqStateCase := 10; 
			END_IF
      
    10: // Nest 2-4 engine stop
      IF TRUE 
			AND THIS^.itfNest2.M_StopEngine()
			AND THIS^.itfNest3.M_StopEngine()
			AND THIS^.itfNest4.M_StopEngine()
			THEN 
				THIS^.stSeqCtrlGeneral.iInternalSeqStateCase := 1000; 
			END_IF
      
    1000: // Exit step
      IF TRUE
      AND THIS^.itfTimerNest1.M_StopTimer()
      AND THIS^.itfTimerNest2.M_StopTimer()
      AND THIS^.itfTimerNest3.M_StopTimer()
      AND THIS^.itfTimerNest4.M_StopTimer()
			THEN 
				THIS^.stSeqCtrlGeneral.iInternalSeqStateCase := 9999; 
			END_IF
      
	ELSE
		THIS^.stSeqCtrlGeneral.eActiveSeqState := E_SEQ_GENERAL.DONE;  
	END_CASE
	THIS^.stSeqCtrlGeneral.strExtraInfo := CONCAT('Internal state: ', TO_STRING(THIS^.stSeqCtrlGeneral.iInternalSeqStateCase));
E_SEQ_GENERAL.DONE:;
E_SEQ_GENERAL.ERROR:;
E_SEQ_GENERAL.TIME_OUT:; 

IF TRUE
AND THIS^.stSeqCtrlGeneral.bTimeOutActiveQuit 
THEN
  THIS^.stSeqCtrlGeneral.strExtraInfo := 'Bitte quittieren und erneut testen';
  IF TRUE
  //AND itfOpMode.P_QUIT
  THEN
    THIS^.stSeqCtrlGeneral.eActiveSeqState := E_SEQ_GENERAL.EXECUTE;
	END_IF
  
END_IF

ELSE
  THIS^.stSeqCtrlGeneral.eActiveSeqState := E_SEQ_GENERAL.ERROR;
END_CASE
END_METHOD

METHOD PRIVATE _m_SequenceManager
VAR_INPUT
END_VAR
IF FALSE
//AND THIS^.eActiveSeqState=DONE 
AND eLastSeq<>eSeq
THEN
	IF THIS^.stSeqCtrlGeneral.eActiveSeqState<>E_SEQ_GENERAL.EXECUTE THEN
		THIS^.stSeqCtrlGeneral.eActiveSeqState:=E_SEQ_GENERAL.READY;
	END_IF
END_IF

eSeq := eNextSeq;

//DelayTimer und TimeOut Timer verwalten
stSeqCtrlGeneral.bActiveStep:=	TRUE
				AND eLastSeq					=	eSeq
				AND stSeqCtrlGeneral.eLastActiveSeqState			=	stSeqCtrlGeneral.eActiveSeqState
				AND	stSeqCtrlGeneral.iLastInternalSeqStateCase	=	stSeqCtrlGeneral.iInternalSeqStateCase
				;
			
IF NOT stSeqCtrlGeneral.bActiveStep THEN
	stSeqCtrlGeneral.bDelayActive:=FALSE;
	stSeqCtrlGeneral.bTimeOutActiveQuit:=FALSE;
	stSeqCtrlGeneral.bTimeOutActiveNoQuit:=FALSE;
  THIS^.stSeqCtrlGeneral.strExtraInfo:='';
END_IF

_m_SaveLastStep();
stSeqCtrlGeneral.tonDelay	(IN:=stSeqCtrlGeneral.bActiveStep AND stSeqCtrlGeneral.bDelayActive, 		PT:=stSeqCtrlGeneral.tDelay);
stSeqCtrlGeneral.tonTimeOut	(IN:=stSeqCtrlGeneral.bActiveStep AND (stSeqCtrlGeneral.bTimeOutActiveNoQuit OR stSeqCtrlGeneral.bTimeOutActiveQuit), 	PT:=stSeqCtrlGeneral.tTimeOut);
stSeqCtrlGeneral.tonStepTime	(IN:= stSeqCtrlGeneral.bActiveStep, PT:= T#24H);

IF stSeqCtrlGeneral.tonTimeOut.Q  THEN
	stSeqCtrlGeneral.eActiveSeqState:=E_SEQ_GENERAL.TIME_OUT;
END_IF

IF stSeqCtrlGeneral.iError<>0 THEN
	eSeq:=E_SEQ_PROCESS.ERROR_SEQ;
END_IF



eLastSeq					:=	eSeq;
stSeqCtrlGeneral.eLastActiveSeqState			:=	stSeqCtrlGeneral.eActiveSeqState;
stSeqCtrlGeneral.iLastInternalSeqStateCase	:=	stSeqCtrlGeneral.iInternalSeqStateCase;

// Reset set ready state
IF THIS^.stSeqCtrlGeneral.bExitSetReadyState THEN
  THIS^.stSeqCtrlGeneral.bExitSetReadyState := FALSE;
END_IF
END_METHOD

METHOD PRIVATE _m_TimeOut : BOOL
VAR_INPUT
	bTimeoutActiveToQuit:	BOOL;
	bTimeOutActiveNoQuit:	BOOL;
	tTimeOut:				TIME;	
END_VAR
THIS^.stSeqCtrlGeneral.bTimeOutActiveQuit:=	bTimeoutActiveToQuit;
THIS^.stSeqCtrlGeneral.bTimeOutActiveNoQuit:=	bTimeOutActiveNoQuit;
THIS^.stSeqCtrlGeneral.tTimeOut:=			tTimeOut;
_m_TimeOut:=FALSE;
IF THIS^.stSeqCtrlGeneral.tonTimeOut.Q THEN
	_m_TimeOut:=TRUE;
END_IF
END_METHOD

METHOD FB_init : BOOL
VAR_INPUT
	bInitRetains : BOOL; // if TRUE, the retain variables are initialized (warm start / cold start)
	bInCopyCode : BOOL;  // if TRUE, the instance afterwards gets moved into the copy code (online change)
  
  itfLogEvents: 										                      I_HANDLE_EVENTS;
  itfOpMode:											                        I_OP_MODE; 
  itfTimerNest1:                                          I_CLOCK; 
  itfTimerNest2:                                          I_CLOCK; 
  itfTimerNest3:                                          I_CLOCK; 
  itfTimerNest4:                                          I_CLOCK;
  itfNest1:                                               I_PROCESS_NEST1;
  itfNest2:                                               I_PROCESS_NEST2_4;
  itfNest3:                                               I_PROCESS_NEST2_4;
  itfNest4:                                               I_PROCESS_NEST2_4;
  itfLowPressurePump:                                     I_PUMP_WITH_BYPASS;
  itfOilCooler:                                           I_PUMP;
  itfBypassPump:                                          I_PUMP;
  itfLevelSwitch_AggregateTank1_Out1:                     I_BINARY_SWITCH;
  itfLevelSwitch_AggregateTank1_Out2:                     I_BINARY_SWITCH;
  itfTemperatureSwitch_AggregateTank1_Out1:               I_BINARY_SWITCH;
  itfTemperatureSwitch_AggregateTank1_Out2:               I_BINARY_SWITCH;
  itfLevelSwitch_AggregateTank2_Out1:                     I_BINARY_SWITCH;
  itfLevelSwitch_AggregateTank2_Out2:                     I_BINARY_SWITCH;
  itfLevelSwitch_AggregateTank2_Out3:                     I_BINARY_SWITCH;
  itfSwitch_AggregateFilter_Dirty:                        I_BINARY_SWITCH; 
END_VAR
THIS^.itfLogEvents := itfLogEvents;
THIS^.itfOpMode := itfOpMode;
THIS^.itfTimerNest1 := itfTimerNest1;
THIS^.itfTimerNest2 := itfTimerNest2;
THIS^.itfTimerNest3 := itfTimerNest3;
THIS^.itfTimerNest4 := itfTimerNest4;
THIS^.itfNest1 := itfNest1;
THIS^.itfNest2 := itfNest2;
THIS^.itfNest3 := itfNest3;
THIS^.itfNest4 := itfNest4;
THIS^.itfLowPressurePump := itfLowPressurePump;
THIS^.itfOilCooler := itfOilCooler;
THIS^.itfBypassPump := itfBypassPump;
THIS^.itfLevelSwitch_AggregateTank1_Out1 := itfLevelSwitch_AggregateTank1_Out1;
THIS^.itfLevelSwitch_AggregateTank1_Out2 := itfLevelSwitch_AggregateTank1_Out2;
THIS^.itfTemperatureSwitch_AggregateTank1_Out1 := itfTemperatureSwitch_AggregateTank1_Out1;
THIS^.itfTemperatureSwitch_AggregateTank1_Out2 := itfTemperatureSwitch_AggregateTank1_Out2;
THIS^.itfLevelSwitch_AggregateTank2_Out1 := itfLevelSwitch_AggregateTank2_Out1;
THIS^.itfLevelSwitch_AggregateTank2_Out2 := itfLevelSwitch_AggregateTank2_Out2;
THIS^.itfLevelSwitch_AggregateTank2_Out3 := itfLevelSwitch_AggregateTank2_Out3;
THIS^.itfSwitch_AggregateFilter_Dirty := itfSwitch_AggregateFilter_Dirty;
END_METHOD

METHOD M_BreakPressureDet : BOOL
VAR_INPUT
  stBreakPressureParams:                 ST_RECIPE_BREAK_PRESSURE;
END_VAR
M_BreakPressureDet := THIS^.stSeqCtrlGeneral.eActiveSeqState = E_SEQ_GENERAL.DONE;

// Assign input
THIS^.stBPDParams := stBreakPressureParams;

// General
IF THIS^.stSeqCtrlGeneral.eActiveSeqState = E_SEQ_GENERAL.READY THEN
  THIS^.eNextSeq := E_SEQ_PROCESS.BREAK_PRESSURE_DET;
  THIS^.stSeqCtrlGeneral.eActiveSeqState := E_SEQ_GENERAL.EXECUTE;
END_IF
END_METHOD

METHOD M_EnduranceRun : BOOL
VAR_INPUT
  stEnduranceRunParams:                 ST_RECIPE_ENDURANCE_RUN;
END_VAR
M_EnduranceRun := THIS^.stSeqCtrlGeneral.eActiveSeqState = E_SEQ_GENERAL.DONE;

// Assign input
THIS^.stERParams := stEnduranceRunParams;

// General
IF THIS^.stSeqCtrlGeneral.eActiveSeqState = E_SEQ_GENERAL.READY THEN
  THIS^.eNextSeq := E_SEQ_PROCESS.ENDURANCE_RUN;
  THIS^.stSeqCtrlGeneral.eActiveSeqState := E_SEQ_GENERAL.EXECUTE;
END_IF
END_METHOD

METHOD M_EStop : BOOL
M_EStop := THIS^.stSeqCtrlGeneral.eActiveSeqState = E_SEQ_GENERAL.DONE;

IF THIS^.stSeqCtrlGeneral.eActiveSeqState = E_SEQ_GENERAL.READY THEN
  THIS^.eNextSeq := E_SEQ_PROCESS.ESTOP;
  THIS^.stSeqCtrlGeneral.eActiveSeqState := E_SEQ_GENERAL.EXECUTE;
END_IF
END_METHOD

METHOD M_LeakTest1 : BOOL
VAR_INPUT
  stLeakTest1Params:                 ST_RECIPE_LEAK_TEST1;
END_VAR
M_LeakTest1 := THIS^.stSeqCtrlGeneral.eActiveSeqState = E_SEQ_GENERAL.DONE;

// Assign input
THIS^.stLT1Params := stLeakTest1Params;

// General
IF THIS^.stSeqCtrlGeneral.eActiveSeqState = E_SEQ_GENERAL.READY THEN
  THIS^.eNextSeq := E_SEQ_PROCESS.LEAK_TEST_1;
  THIS^.stSeqCtrlGeneral.eActiveSeqState := E_SEQ_GENERAL.EXECUTE;
END_IF
END_METHOD

METHOD M_LeakTest2 : BOOL
VAR_INPUT
  stLeakTest2Params:                 ST_RECIPE_LEAK_TEST2;
END_VAR
M_LeakTest2 := THIS^.stSeqCtrlGeneral.eActiveSeqState = E_SEQ_GENERAL.DONE;

// Assign input
THIS^.stLT2Params := stLeakTest2Params;

// General
IF THIS^.stSeqCtrlGeneral.eActiveSeqState = E_SEQ_GENERAL.READY THEN
  THIS^.eNextSeq := E_SEQ_PROCESS.LEAK_TEST_2;
  THIS^.stSeqCtrlGeneral.eActiveSeqState := E_SEQ_GENERAL.EXECUTE;
END_IF
END_METHOD

METHOD M_Reset : BOOL
M_Reset := THIS^.stSeqCtrlGeneral.eActiveSeqState = E_SEQ_GENERAL.DONE;

IF THIS^.stSeqCtrlGeneral.eActiveSeqState = E_SEQ_GENERAL.READY THEN
  THIS^.eNextSeq := E_SEQ_PROCESS.INIT;
  THIS^.stSeqCtrlGeneral.eActiveSeqState := E_SEQ_GENERAL.EXECUTE;
END_IF
END_METHOD

{warning 'Methodenimplementierung hinzufügen'}
(*=== Method: M_Run  ============================================

 @brief: Here is the global code (Timer, Event, Flange,...)*)
METHOD M_Run
END_METHOD

METHOD M_SetReady : BOOL
VAR_INPUT
  
END_VAR
M_SetReady := TRUE
              AND THIS^.stSeqCtrlGeneral.eActiveSeqState = E_SEQ_GENERAL.READY
              AND THIS^.eSeq = E_SEQ_PROCESS.BASE;

THIS^.stSeqCtrlGeneral.eActiveSeqState := E_SEQ_GENERAL.READY;
THIS^.eNextSeq := E_SEQ_PROCESS.BASE;
END_METHOD

METHOD M_Stop : BOOL
M_Stop := THIS^.stSeqCtrlGeneral.eActiveSeqState = E_SEQ_GENERAL.DONE;

IF THIS^.stSeqCtrlGeneral.eActiveSeqState = E_SEQ_GENERAL.READY THEN
  THIS^.eNextSeq := E_SEQ_PROCESS.STOP;
  THIS^.stSeqCtrlGeneral.eActiveSeqState := E_SEQ_GENERAL.EXECUTE;
END_IF
END_METHOD

METHOD M_StopEngine : BOOL
M_StopEngine := THIS^.stSeqCtrlGeneral.eActiveSeqState = E_SEQ_GENERAL.DONE;

IF THIS^.stSeqCtrlGeneral.eActiveSeqState = E_SEQ_GENERAL.READY THEN
  THIS^.eNextSeq := E_SEQ_PROCESS.STOP_ENGINE;
  THIS^.stSeqCtrlGeneral.eActiveSeqState := E_SEQ_GENERAL.EXECUTE;
END_IF
END_METHOD

{warning 'Eigenschaftenimplementierung hinzufügen'}
PROPERTY P_CurrentCycleNest1 : UDINT
GET
P_CurrentCycleNest1 := THIS^.udiCurrentCyclesNest1;
END_GET
END_PROPERTY

{warning 'Eigenschaftenimplementierung hinzufügen'}
PROPERTY P_CurrentCycleNest2 : UDINT
GET
P_CurrentCycleNest2 := THIS^.udiCurrentCyclesNest2;
END_GET
END_PROPERTY

{warning 'Eigenschaftenimplementierung hinzufügen'}
PROPERTY P_CurrentCycleNest3 : UDINT
GET
P_CurrentCycleNest3 := THIS^.udiCurrentCyclesNest3;
END_GET
END_PROPERTY

{warning 'Eigenschaftenimplementierung hinzufügen'}
PROPERTY P_CurrentCycleNest4 : UDINT
GET
P_CurrentCycleNest4 := THIS^.udiCurrentCyclesNest4;
END_GET
END_PROPERTY

{warning 'Eigenschaftenimplementierung hinzufügen'}
(*=== Property: P_Event  ============================================

 @param [set]: 	Set the Structure "ST_EVENT" from another Object
 @param [get]: 	Return the Structure "ST_EVENT", it contains the actual 
					event of the Object *)
PROPERTY P_Event : GenLib.ST_EVENT
GET
END_GET
SET
END_SET
END_PROPERTY

{warning 'Eigenschaftenimplementierung hinzufügen'}
(*=== Property: P_FullObjectPath  ============================================

 @param [set]: 	Set the Object Path (Clear String of Object)
 @param [get]: 	Return the Objectpath *)
PROPERTY P_FullObjectPath : STRING
GET
END_GET
SET
END_SET
END_PROPERTY

{warning 'Eigenschaftenimplementierung hinzufügen'}
(*=== Property: P_Global_Ack  ============================================

 @param [set]: 	Set the Bit for Ack from another Object
 @param [get]: 	Return the state of Ack Bit*)
PROPERTY P_Global_Ack : BOOL
GET
END_GET
SET
END_SET
END_PROPERTY

{warning 'Eigenschaftenimplementierung hinzufügen'}
(*=== Property: P_GlobalID  ============================================

 @param [set]: 	-
 @param [get]: 	Return the string of instance path*)
PROPERTY P_GlobalID : STRING
GET
END_GET
END_PROPERTY

{warning 'Eigenschaftenimplementierung hinzufügen'}
PROPERTY P_ReadyState : BOOL
GET
P_ReadyState := THIS^.stSeqCtrlGeneral.eActiveSeqState = E_SEQ_GENERAL.READY;
END_GET
END_PROPERTY

END_FUNCTION_BLOCK

(* stored: Version 1.1.0.1, ProductVersion 3.1.4024.12
   POU FB_PROCESS_MAIN: Id {7cea8bf1-c942-49b5-be8f-3059d77d0bfb}, SpecialFunc None
   Folder PRIVAT: Id {5b81d2fd-964a-43ad-80af-f20644ca0ca7}
   Folder SEQUENCE: Id {7916f48d-8930-4ced-8021-94cad8983fbd}
   Method _m_DebugManager: Id {cf40ed13-ecb8-488c-9826-2a9fb2bbbe22}
   Method _m_Delay: Id {9fe78e97-b7f1-4694-8030-974e38869d9d}
   Method _m_GeneralStepSetting: Id {085f52dd-c1bc-4ea3-841f-02b2a510942d}
   Method _m_SaveLastStep: Id {cbf8e374-5358-4576-a72b-39ed2c88550a}
   Method _m_Seq_BREAK_PRESSURE_DET: Id {803e8cfc-fac8-4871-bef3-a56c59b2dfc2}
   Method _m_Seq_ENDURANCE_RUN: Id {a51c6301-7ef0-40f1-b6cb-e2d4dba9ea6c}
   Method _m_Seq_ESTOP: Id {7cd5e55a-1c92-4d0d-a777-74969a94b9eb}
   Method _m_Seq_INIT: Id {22d19214-d003-4baa-8685-e1f60bb1b381}
   Method _m_Seq_LEAK_TEST_1: Id {d8135877-78f7-40cb-9da4-48eea49eacc4}
   Method _m_Seq_LEAK_TEST_2: Id {28208dc8-5c90-40ca-957a-fece5d6f3bfa}
   Method _m_Seq_STOP: Id {1c3b4e49-e1af-4e25-a142-5ab9459cc41c}
   Method _m_Seq_STOP_ENGINE: Id {5cc2e1d3-ed47-4639-85ee-c7eab0e56261}
   Method _m_SequenceManager: Id {e7136404-aa05-42ec-a315-90d24e0aa4b8}
   Method _m_TimeOut: Id {954056a7-9b1a-46fe-a1fd-1a17b3e12e91}
   Method FB_init: Id {c58c5cdc-e298-464a-b4fb-8ebea23b6eb0}
   Method M_BreakPressureDet: Id {3a19c7cb-e4cb-4e98-a0d4-824726720bdb}
   Method M_EnduranceRun: Id {4f2c985e-a721-4788-8160-b7bd44014e33}
   Method M_EStop: Id {a9af6422-b5f6-41c3-b941-cba0672c80e1}
   Method M_LeakTest1: Id {2d6e9442-3e13-407a-ad19-039c1458a116}
   Method M_LeakTest2: Id {74e78652-5781-41e2-97f7-bd6978a0aa80}
   Method M_Reset: Id {b1d69d5b-a763-4801-8d63-7c4d526c8d90}
   Method M_Run: Id {e244540b-5d3f-4fbd-9700-2e295c4229e0}
   Method M_SetReady: Id {deeebce7-d5bd-4f24-8c16-95acf333c335}
   Method M_Stop: Id {1ec4bc67-66b8-4650-a6c2-95be9de96754}
   Method M_StopEngine: Id {a35c34b5-fdcc-401f-b531-82b6bdf8cb6b}
   Property P_CurrentCycleNest1: Id {131e9b6f-9049-4b03-85c5-bd9439f3fb6a}
   Get Get: Id {5e97c001-6589-4db5-957b-66aee716381e}
   Property P_CurrentCycleNest2: Id {9482527d-9936-4eb1-b052-fc636235b448}
   Get Get: Id {af54279a-7608-4a72-8a8d-e1543aadace6}
   Property P_CurrentCycleNest3: Id {8e6ae9c9-9823-4d3f-979f-127298c241b5}
   Get Get: Id {f48f7b80-78b8-4155-ae6d-3cd1e990c593}
   Property P_CurrentCycleNest4: Id {55490af6-5db3-45a7-9ad0-6df259631363}
   Get Get: Id {831bacf7-ee9d-48a7-8745-11bad436360e}
   Property P_Event: Id {6bf2a264-2653-4937-8a4a-e49e7c3b4fef}
   Get Get: Id {9782cbbc-68ac-44e1-bb61-6227f0289d5f}
   Set Set: Id {c310aa41-0c71-48c4-9523-cece13f113d0}
   Property P_FullObjectPath: Id {fa827b5c-2969-4ff3-9db8-9a32eb21cf85}
   Get Get: Id {8b3b202f-c8de-46c2-802d-7bda7bad1cf1}
   Set Set: Id {ed15d441-87ea-4579-8b8c-c77e9fe0d759}
   Property P_Global_Ack: Id {b2d501da-d1c6-4ae5-a5de-bddde3f29458}
   Get Get: Id {ff082c76-7e0a-4698-af2d-cb3d887f45d5}
   Set Set: Id {71248a13-403d-44ca-bfcd-079961348436}
   Property P_GlobalID: Id {998d72c3-2a3f-453c-beef-42fe3234a473}
   Get Get: Id {83200a4d-999f-40e1-a2fa-d827af50c480}
   Property P_ReadyState: Id {a5a914d2-6d93-4ec4-9867-3bbf7d8f3310}
   Get Get: Id {ade13aa0-502f-44c6-8ec7-aea56933f6cc} *)
